Staubli VAL3: Valve.pgx

program Valve(bool cde)
begin
  //*******************************************************************************
  //*   ______
  //*  / _____) /|
  //* | |      / /
  //* | | /\  / /
  //* | | \ \/ /  _      Copyright (c) KEOLABS, 2016
  //* | |  \__/  | |        http://www.keolabs.com
  //* | |________| |
  //*  \__________/
  //*
  //********************************************************************************
  //*@file          : Valve
  //*@author        : Yves Ragot
  //*@version       : $Id: Valve.pgx 1882 2019-01-10 16:18:45Z xavier $
  //*@brief         : Valve command
  //*
  //*******************************************************************************/

  //valve1 = cde
  if (cde)
    open(tCurrentTool)
  else
    close(tCurrentTool)
  endIf

end
